// Mitsubishi GX Developer project: tocco20140630画像   PLC: FX1N

PROGRAM MAIN
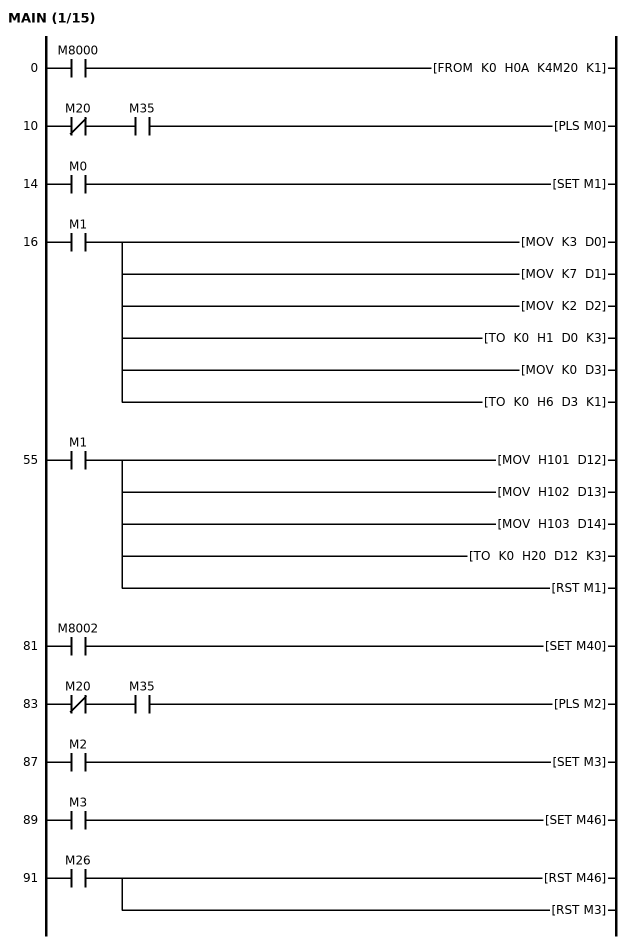
0     LD      M8000
      FROM    K0 H0A K4M20 K1
10    LDI     M20
      AND     M35
      PLS     M0
14    LD      M0
      SET     M1
16    LD      M1
      MOV     K3 D0
      MOV     K7 D1
      MOV     K2 D2
      TO      K0 H1 D0 K3
      MOV     K0 D3
      TO      K0 H6 D3 K1
55    LD      M1
      MOV     H101 D12
      MOV     H102 D13
      MOV     H103 D14
      TO      K0 H20 D12 K3
      RST     M1
81    LD      M8002
      SET     M40
83    LDI     M20
      AND     M35
      PLS     M2
87    LD      M2
      SET     M3
89    LD      M3
      SET     M46
91    LD      M26
      RST     M46
      RST     M3
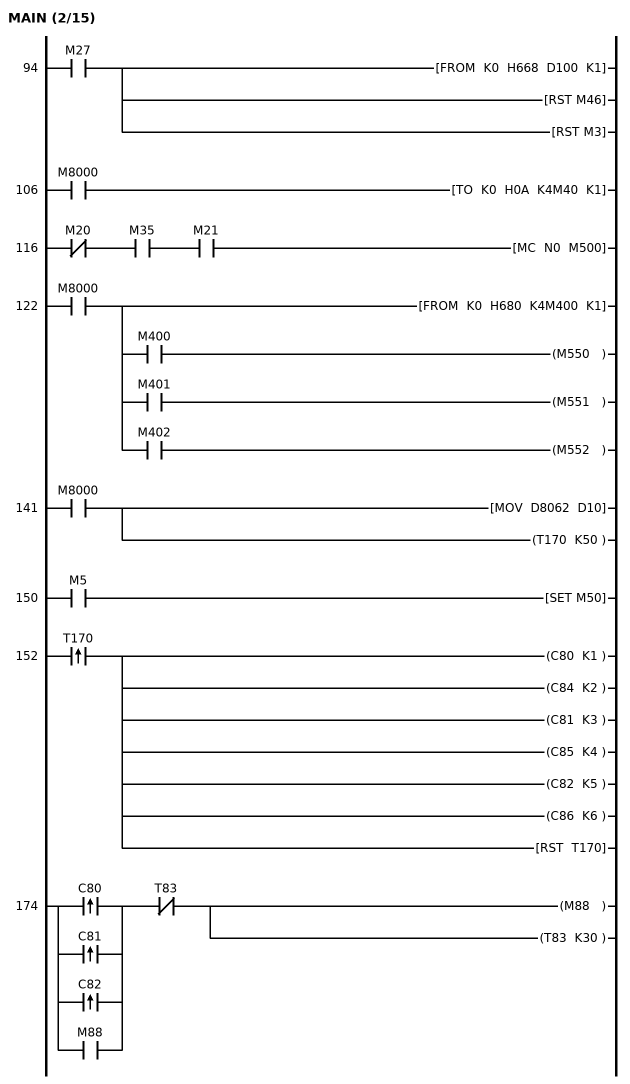
94    LD      M27
      FROM    K0 H668 D100 K1
      RST     M46
      RST     M3
106   LD      M8000
      TO      K0 H0A K4M40 K1
116   LDI     M20
      AND     M35
      AND     M21
      MC      N0 M500
122   LD      M8000
      FROM    K0 H680 K4M400 K1
      MPS
      AND     M400
      OUT     M550
      MRD
      AND     M401
      OUT     M551
      MPP
      AND     M402
      OUT     M552
141   LD      M8000
      MOV     D8062 D10
      OUT     T170 K50
150   LD      M5
      SET     M50
152   LDP     T170
      OUT     C80 K1
      OUT     C84 K2
      OUT     C81 K3
      OUT     C85 K4
      OUT     C82 K5
      OUT     C86 K6
      RST     T170
174   LDP     C80
      ORP     C81
      ORP     C82
      OR      M88
      ANI     T83
      OUT     M88
      OUT     T83 K30
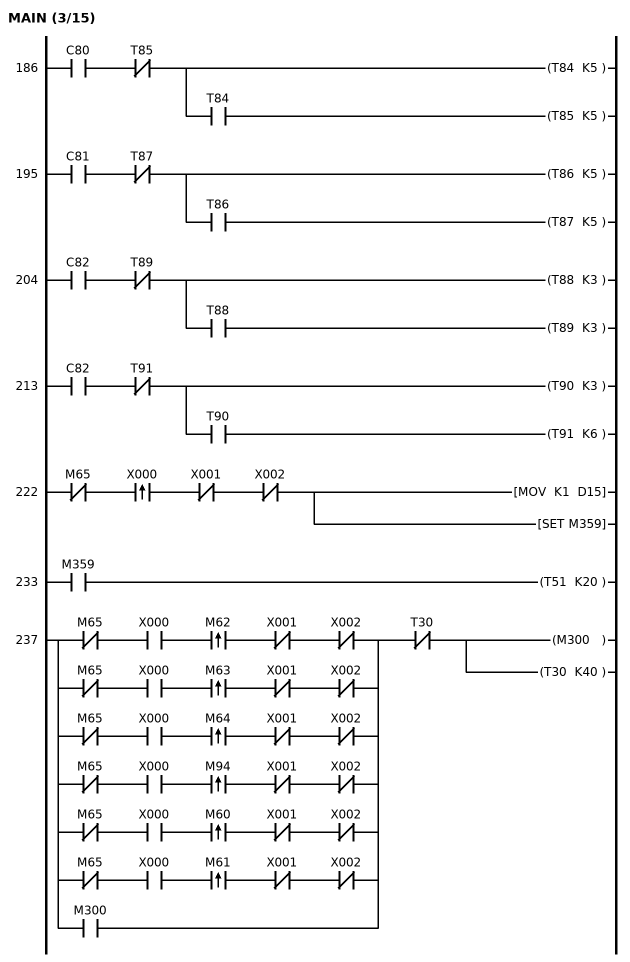
186   LD      C80
      ANI     T85
      OUT     T84 K5
      AND     T84
      OUT     T85 K5
195   LD      C81
      ANI     T87
      OUT     T86 K5
      AND     T86
      OUT     T87 K5
204   LD      C82
      ANI     T89
      OUT     T88 K3
      AND     T88
      OUT     T89 K3
213   LD      C82
      ANI     T91
      OUT     T90 K3
      AND     T90
      OUT     T91 K6
222   LDI     M65
      ANDP    X000
      ANI     X001
      ANI     X002
      MOV     K1 D15
      SET     M359
233   LD      M359
      OUT     T51 K20
237   LDI     M65
      AND     X000
      ANDP    M62
      ANI     X001
      ANI     X002
      LDI     M65
      AND     X000
      ANDP    M63
      ANI     X001
      ANI     X002
      ORB
      LDI     M65
      AND     X000
      ANDP    M64
      ANI     X001
      ANI     X002
      ORB
      LDI     M65
      AND     X000
      ANDP    M94
      ANI     X001
      ANI     X002
      ORB
      LDI     M65
      AND     X000
      ANDP    M60
      ANI     X001
      ANI     X002
      ORB
      LDI     M65
      AND     X000
      ANDP    M61
      ANI     X001
      ANI     X002
      ORB
      OR      M300
      ANI     T30
      OUT     M300
      OUT     T30 K40
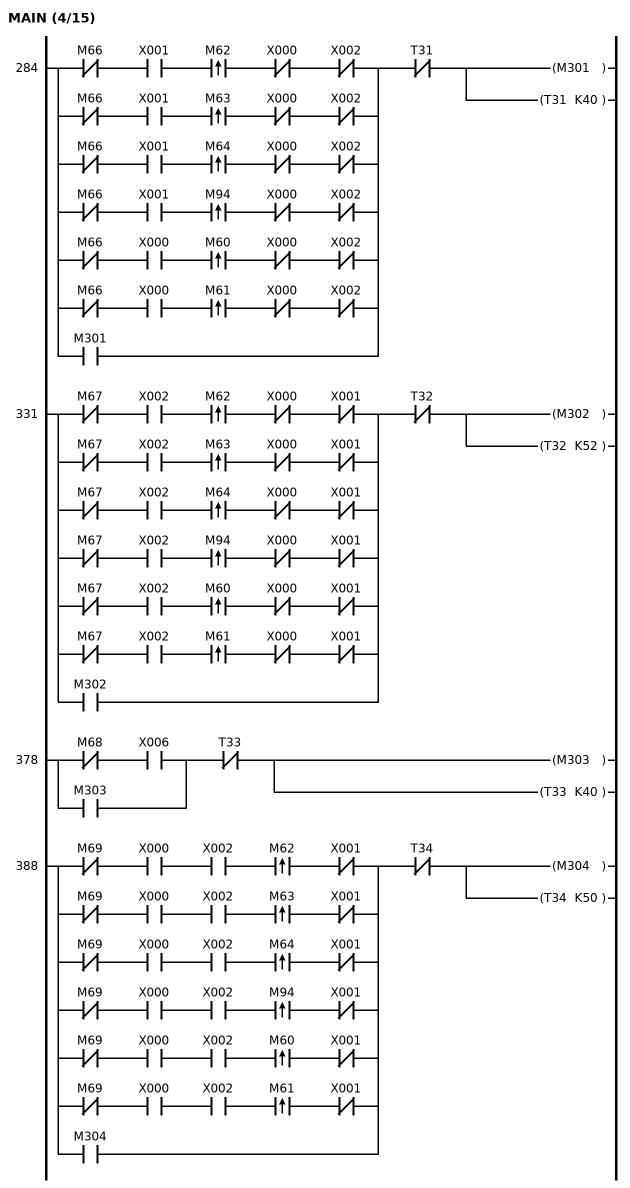
284   LDI     M66
      AND     X001
      ANDP    M62
      ANI     X000
      ANI     X002
      LDI     M66
      AND     X001
      ANDP    M63
      ANI     X000
      ANI     X002
      ORB
      LDI     M66
      AND     X001
      ANDP    M64
      ANI     X000
      ANI     X002
      ORB
      LDI     M66
      AND     X001
      ANDP    M94
      ANI     X000
      ANI     X002
      ORB
      LDI     M66
      AND     X000
      ANDP    M60
      ANI     X000
      ANI     X002
      ORB
      LDI     M66
      AND     X000
      ANDP    M61
      ANI     X000
      ANI     X002
      ORB
      OR      M301
      ANI     T31
      OUT     M301
      OUT     T31 K40
331   LDI     M67
      AND     X002
      ANDP    M62
      ANI     X000
      ANI     X001
      LDI     M67
      AND     X002
      ANDP    M63
      ANI     X000
      ANI     X001
      ORB
      LDI     M67
      AND     X002
      ANDP    M64
      ANI     X000
      ANI     X001
      ORB
      LDI     M67
      AND     X002
      ANDP    M94
      ANI     X000
      ANI     X001
      ORB
      LDI     M67
      AND     X002
      ANDP    M60
      ANI     X000
      ANI     X001
      ORB
      LDI     M67
      AND     X002
      ANDP    M61
      ANI     X000
      ANI     X001
      ORB
      OR      M302
      ANI     T32
      OUT     M302
      OUT     T32 K52
378   LDI     M68
      AND     X006
      OR      M303
      ANI     T33
      OUT     M303
      OUT     T33 K40
388   LDI     M69
      AND     X000
      AND     X002
      ANDP    M62
      ANI     X001
      LDI     M69
      AND     X000
      AND     X002
      ANDP    M63
      ANI     X001
      ORB
      LDI     M69
      AND     X000
      AND     X002
      ANDP    M64
      ANI     X001
      ORB
      LDI     M69
      AND     X000
      AND     X002
      ANDP    M94
      ANI     X001
      ORB
      LDI     M69
      AND     X000
      AND     X002
      ANDP    M60
      ANI     X001
      ORB
      LDI     M69
      AND     X000
      AND     X002
      ANDP    M61
      ANI     X001
      ORB
      OR      M304
      ANI     T34
      OUT     M304
      OUT     T34 K50
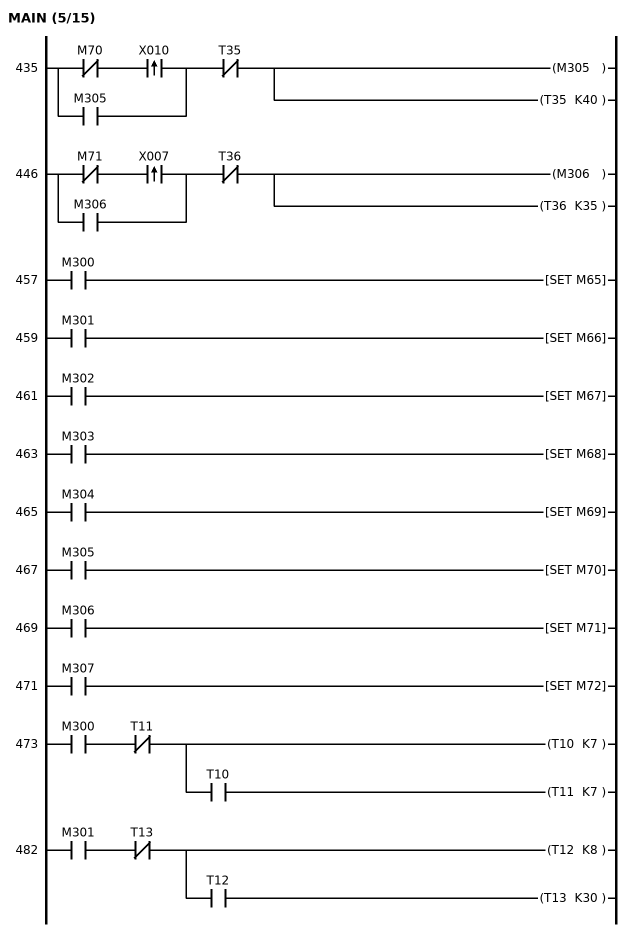
435   LDI     M70
      ANDP    X010
      OR      M305
      ANI     T35
      OUT     M305
      OUT     T35 K40
446   LDI     M71
      ANDP    X007
      OR      M306
      ANI     T36
      OUT     M306
      OUT     T36 K35
457   LD      M300
      SET     M65
459   LD      M301
      SET     M66
461   LD      M302
      SET     M67
463   LD      M303
      SET     M68
465   LD      M304
      SET     M69
467   LD      M305
      SET     M70
469   LD      M306
      SET     M71
471   LD      M307
      SET     M72
473   LD      M300
      ANI     T11
      OUT     T10 K7
      AND     T10
      OUT     T11 K7
482   LD      M301
      ANI     T13
      OUT     T12 K8
      AND     T12
      OUT     T13 K30
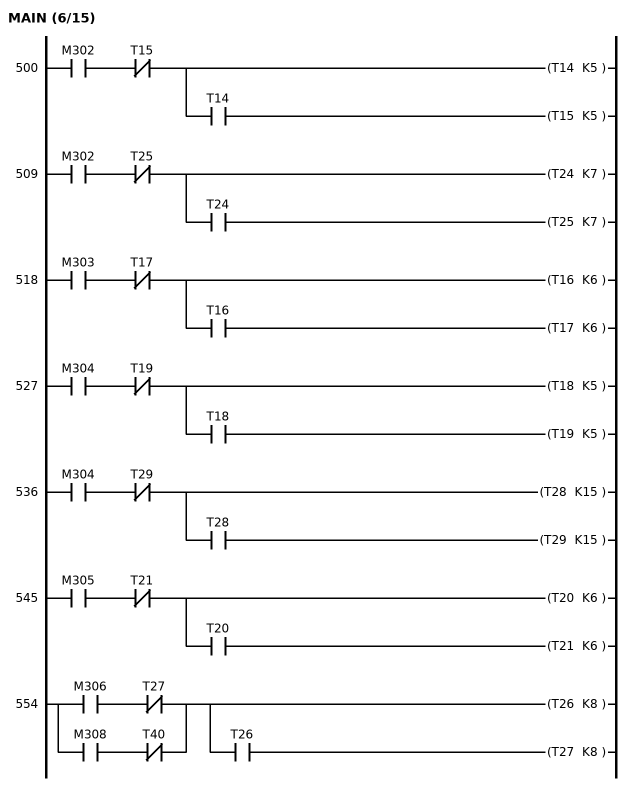
500   LD      M302
      ANI     T15
      OUT     T14 K5
      AND     T14
      OUT     T15 K5
509   LD      M302
      ANI     T25
      OUT     T24 K7
      AND     T24
      OUT     T25 K7
518   LD      M303
      ANI     T17
      OUT     T16 K6
      AND     T16
      OUT     T17 K6
527   LD      M304
      ANI     T19
      OUT     T18 K5
      AND     T18
      OUT     T19 K5
536   LD      M304
      ANI     T29
      OUT     T28 K15
      AND     T28
      OUT     T29 K15
545   LD      M305
      ANI     T21
      OUT     T20 K6
      AND     T20
      OUT     T21 K6
554   LD      M306
      ANI     T27
      LD      M308
      ANI     T40
      ORB
      OUT     T26 K8
      AND     T26
      OUT     T27 K8
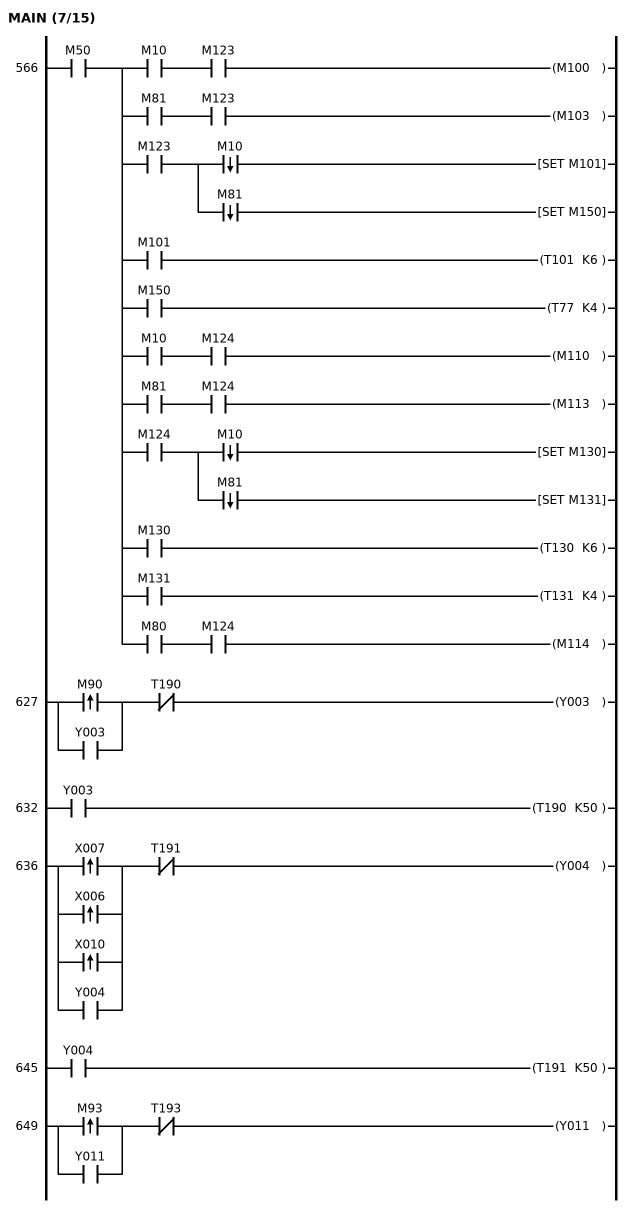
566   LD      M50
      MPS
      AND     M10
      AND     M123
      OUT     M100
      MRD
      AND     M81
      AND     M123
      OUT     M103
      MRD
      AND     M123
      MPS
      ANDF    M10
      SET     M101
      MPP
      ANDF    M81
      SET     M150
      MRD
      AND     M101
      OUT     T101 K6
      MRD
      AND     M150
      OUT     T77 K4
      MRD
      AND     M10
      AND     M124
      OUT     M110
      MRD
      AND     M81
      AND     M124
      OUT     M113
      MRD
      AND     M124
      MPS
      ANDF    M10
      SET     M130
      MPP
      ANDF    M81
      SET     M131
      MRD
      AND     M130
      OUT     T130 K6
      MRD
      AND     M131
      OUT     T131 K4
      MPP
      AND     M80
      AND     M124
      OUT     M114
627   LDP     M90
      OR      Y003
      ANI     T190
      OUT     Y003
632   LD      Y003
      OUT     T190 K50
636   LDP     X007
      ORP     X006
      ORP     X010
      OR      Y004
      ANI     T191
      OUT     Y004
645   LD      Y004
      OUT     T191 K50
649   LDP     M93
      OR      Y011
      ANI     T193
      OUT     Y011
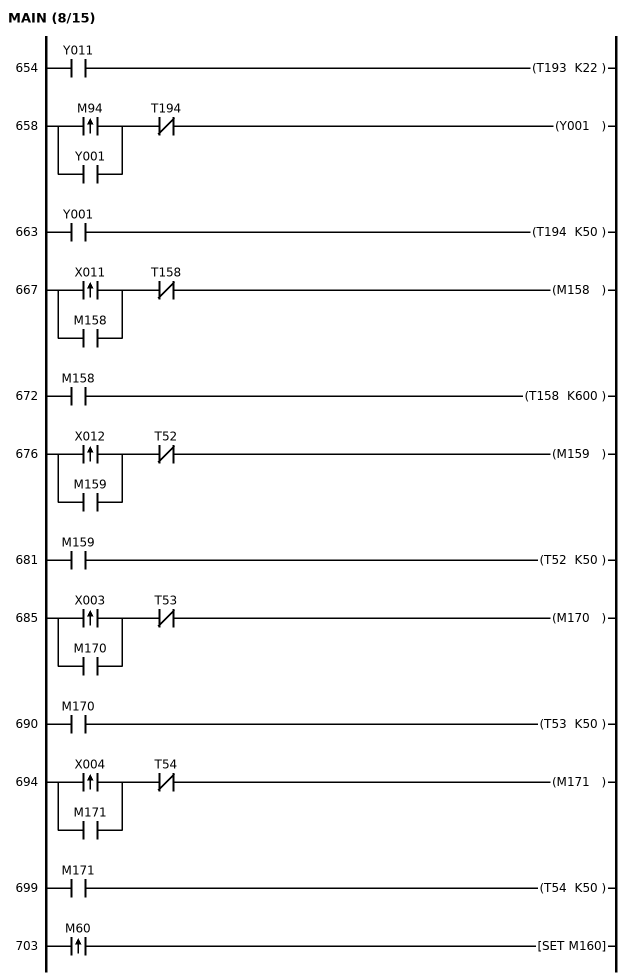
654   LD      Y011
      OUT     T193 K22
658   LDP     M94
      OR      Y001
      ANI     T194
      OUT     Y001
663   LD      Y001
      OUT     T194 K50
667   LDP     X011
      OR      M158
      ANI     T158
      OUT     M158
672   LD      M158
      OUT     T158 K600
676   LDP     X012
      OR      M159
      ANI     T52
      OUT     M159
681   LD      M159
      OUT     T52 K50
685   LDP     X003
      OR      M170
      ANI     T53
      OUT     M170
690   LD      M170
      OUT     T53 K50
694   LDP     X004
      OR      M171
      ANI     T54
      OUT     M171
699   LD      M171
      OUT     T54 K50
703   LDP     M60
      SET     M160
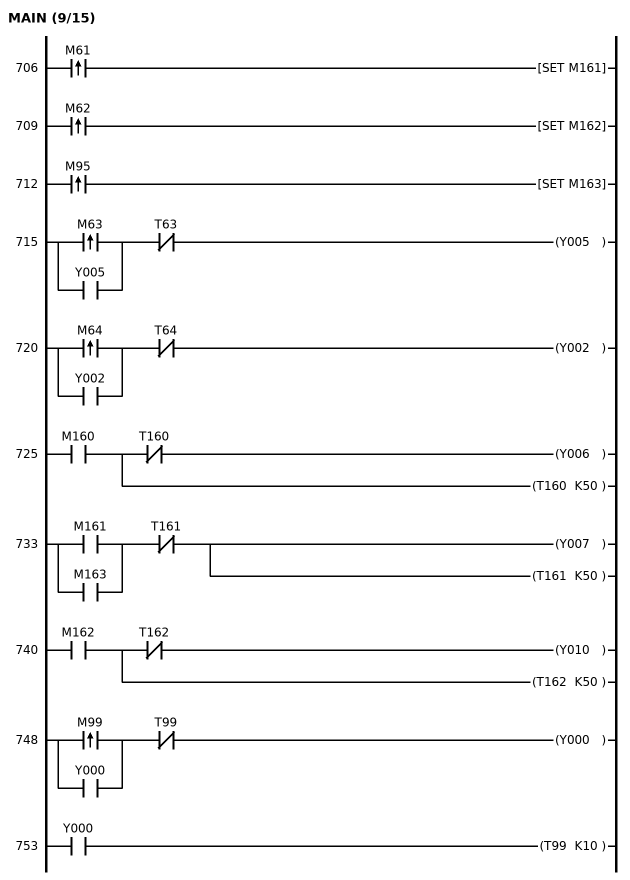
706   LDP     M61
      SET     M161
709   LDP     M62
      SET     M162
712   LDP     M95
      SET     M163
715   LDP     M63
      OR      Y005
      ANI     T63
      OUT     Y005
720   LDP     M64
      OR      Y002
      ANI     T64
      OUT     Y002
725   LD      M160
      MPS
      ANI     T160
      OUT     Y006
      MPP
      OUT     T160 K50
733   LD      M161
      OR      M163
      ANI     T161
      OUT     Y007
      OUT     T161 K50
740   LD      M162
      MPS
      ANI     T162
      OUT     Y010
      MPP
      OUT     T162 K50
748   LDP     M99
      OR      Y000
      ANI     T99
      OUT     Y000
753   LD      Y000
      OUT     T99 K10
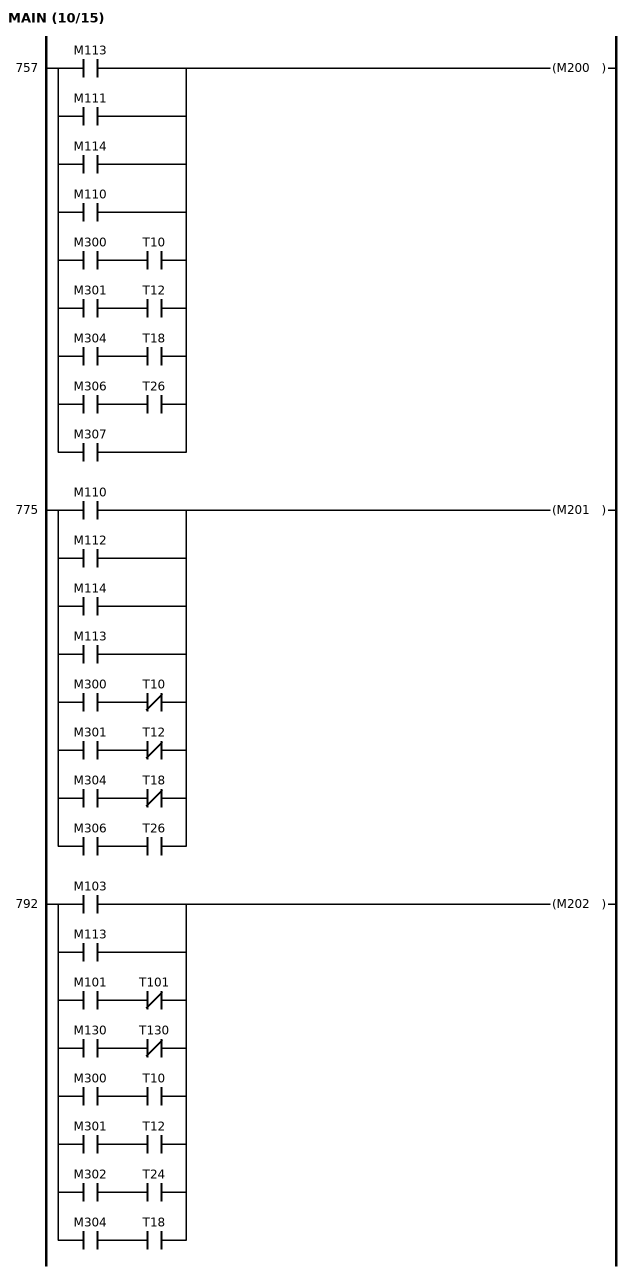
757   LD      M113
      OR      M111
      OR      M114
      OR      M110
      LD      M300
      AND     T10
      ORB
      LD      M301
      AND     T12
      ORB
      LD      M304
      AND     T18
      ORB
      LD      M306
      AND     T26
      ORB
      OR      M307
      OUT     M200
775   LD      M110
      OR      M112
      OR      M114
      OR      M113
      LD      M300
      ANI     T10
      ORB
      LD      M301
      ANI     T12
      ORB
      LD      M304
      ANI     T18
      ORB
      LD      M306
      AND     T26
      ORB
      OUT     M201
792   LD      M103
      OR      M113
      LD      M101
      ANI     T101
      ORB
      LD      M130
      ANI     T130
      ORB
      LD      M300
      AND     T10
      ORB
      LD      M301
      AND     T12
      ORB
      LD      M302
      AND     T24
      ORB
      LD      M304
      AND     T18
      ORB
      OUT     M202
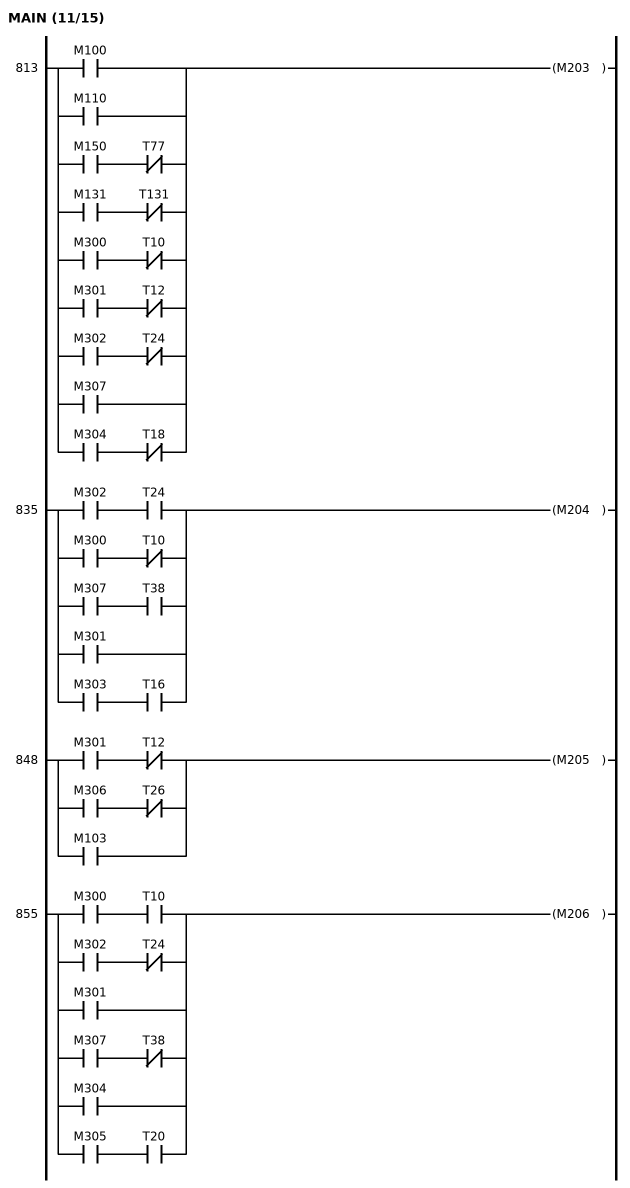
813   LD      M100
      OR      M110
      LD      M150
      ANI     T77
      ORB
      LD      M131
      ANI     T131
      ORB
      LD      M300
      ANI     T10
      ORB
      LD      M301
      ANI     T12
      ORB
      LD      M302
      ANI     T24
      ORB
      OR      M307
      LD      M304
      ANI     T18
      ORB
      OUT     M203
835   LD      M302
      AND     T24
      LD      M300
      ANI     T10
      ORB
      LD      M307
      AND     T38
      ORB
      OR      M301
      LD      M303
      AND     T16
      ORB
      OUT     M204
848   LD      M301
      ANI     T12
      LD      M306
      ANI     T26
      ORB
      OR      M103
      OUT     M205
855   LD      M300
      AND     T10
      LD      M302
      ANI     T24
      ORB
      OR      M301
      LD      M307
      ANI     T38
      ORB
      OR      M304
      LD      M305
      AND     T20
      ORB
      OUT     M206
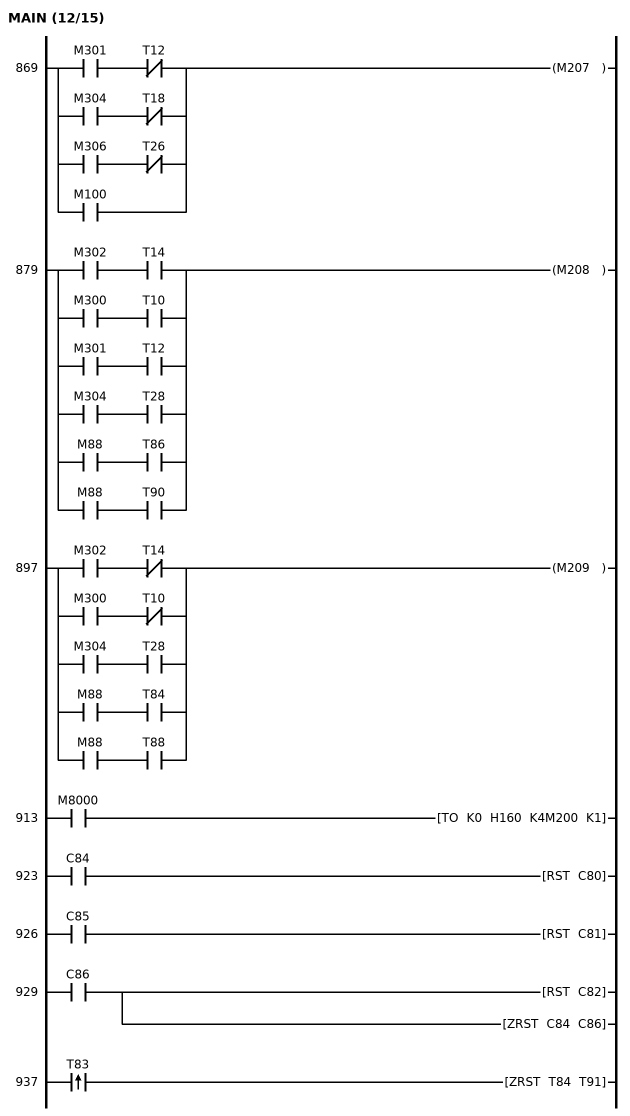
869   LD      M301
      ANI     T12
      LD      M304
      ANI     T18
      ORB
      LD      M306
      ANI     T26
      ORB
      OR      M100
      OUT     M207
879   LD      M302
      AND     T14
      LD      M300
      AND     T10
      ORB
      LD      M301
      AND     T12
      ORB
      LD      M304
      AND     T28
      ORB
      LD      M88
      AND     T86
      ORB
      LD      M88
      AND     T90
      ORB
      OUT     M208
897   LD      M302
      ANI     T14
      LD      M300
      ANI     T10
      ORB
      LD      M304
      AND     T28
      ORB
      LD      M88
      AND     T84
      ORB
      LD      M88
      AND     T88
      ORB
      OUT     M209
913   LD      M8000
      TO      K0 H160 K4M200 K1
923   LD      C84
      RST     C80
926   LD      C85
      RST     C81
929   LD      C86
      RST     C82
      ZRST    C84 C86
937   LDP     T83
      ZRST    T84 T91
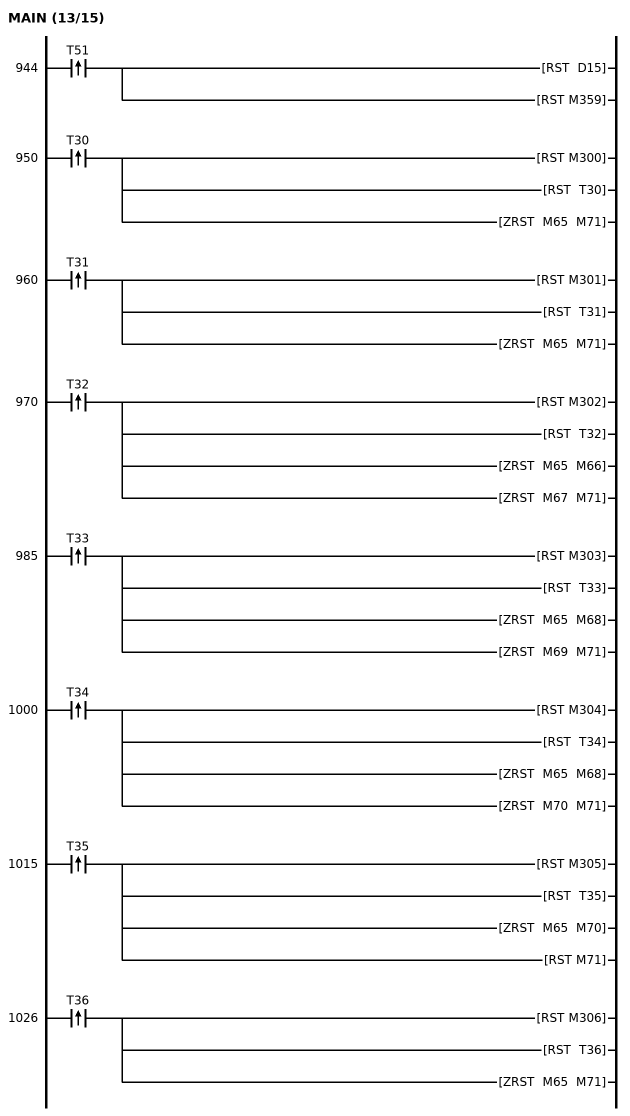
944   LDP     T51
      RST     D15
      RST     M359
950   LDP     T30
      RST     M300
      RST     T30
      ZRST    M65 M71
960   LDP     T31
      RST     M301
      RST     T31
      ZRST    M65 M71
970   LDP     T32
      RST     M302
      RST     T32
      ZRST    M65 M66
      ZRST    M67 M71
985   LDP     T33
      RST     M303
      RST     T33
      ZRST    M65 M68
      ZRST    M69 M71
1000  LDP     T34
      RST     M304
      RST     T34
      ZRST    M65 M68
      ZRST    M70 M71
1015  LDP     T35
      RST     M305
      RST     T35
      ZRST    M65 M70
      RST     M71
1026  LDP     T36
      RST     M306
      RST     T36
      ZRST    M65 M71
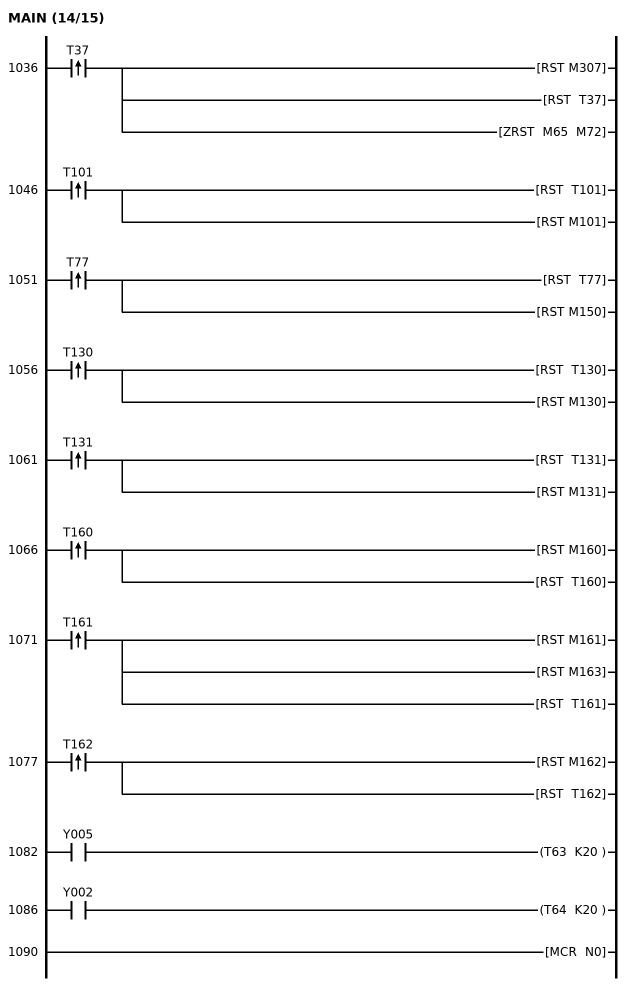
1036  LDP     T37
      RST     M307
      RST     T37
      ZRST    M65 M72
1046  LDP     T101
      RST     T101
      RST     M101
1051  LDP     T77
      RST     T77
      RST     M150
1056  LDP     T130
      RST     T130
      RST     M130
1061  LDP     T131
      RST     T131
      RST     M131
1066  LDP     T160
      RST     M160
      RST     T160
1071  LDP     T161
      RST     M161
      RST     M163
      RST     T161
1077  LDP     T162
      RST     M162
      RST     T162
1082  LD      Y005
      OUT     T63 K20
1086  LD      Y002
      OUT     T64 K20
1090  MCR     N0
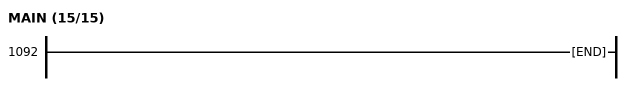
1092  END
END_PROGRAM
